Staubli VAL3: ModelParameter.dtx

public num StiffnessParm[6]
public num DampingParm[6]
public num MassParm[6]
